(* Logix 5000 project; controller Project_Template vendor 1 type 14 code 106 rev 33.12; software revision 33.00 *)

TASK MainTask (continuous, watchdog 500 ms) : MainProgram

MODULES
   Local : vendor 1 type 14 code 106 (Compact 0, rev 33.12)
      Discrete_In_Slot_3 : 1769-IQ16 (Compact 3, rev 1.1, Input RPI 20 ms)
      Discrete_In_Slot_2 : 1769-IQ16 (Compact 2, rev 1.1, Input RPI 20 ms)
      Discrete_Out_Slot_4 : 1769-OW16 (Compact 4, rev 1.1, Output RPI 20 ms)
      ASCII_Slot_1 : vendor 1 type 109 code 66 (Compact 1, rev 2.1, Output RPI 100 ms)
      Discrete_Out_Slot_5 : 1769-OW16 (Compact 5, rev 1.1, Output RPI 20 ms)
END_MODULES

VAR_GLOBAL   (* controller tags *)
   AT_HOME : BOOL;
   AUTO : BOOL;
   end_start : BOOL;
   FLASH_FAST : BOOL := 1;
   Flash_Fast_Off : TIMER := (PRE := 250, ACC := 205, EN := 1, TT := 1);
   Flash_Fast_On : TIMER := (PRE := 250, ACC := 250, EN := 1, DN := 1);
   FLASH_MEDIUM : BOOL := 1;
   Flash_Medium_Off : TIMER := (PRE := 500, ACC := 467, EN := 1, TT := 1);
   Flash_Medium_On : TIMER := (PRE := 500, ACC := 500, EN := 1, DN := 1);
   FLASH_SLOW : BOOL;
   Flash_Slow_Off : TIMER := (PRE := 1000);
   Flash_Slow_On : TIMER := (PRE := 1000, ACC := 957, EN := 1, TT := 1);
   I_Auto_Mode_Selector : ALIAS FOR Local:2:I.Data.2;
   I_Barcode_Stop_Raised : ALIAS FOR Local:3:I.Data.1;
   I_Box_Ejector_Extended : ALIAS FOR Local:2:I.Data.4;
   I_Reject_Cyl_Lowered : ALIAS FOR Local:3:I.Data.2;
   I_Reset_PB : ALIAS FOR Local:2:I.Data.3;
   I_Start_PB : ALIAS FOR Local:2:I.Data.0;
   I_Stop_PB : ALIAS FOR Local:2:I.Data.1;
   I_Vacuum_Head_at_Conveyor : ALIAS FOR Local:3:I.Data.0;
   I_Vacuum_Head_at_Magazine : ALIAS FOR Local:2:I.Data.15;
   I_Vacuum_Head_Extended : ALIAS FOR Local:2:I.Data.14;
   I_Vacuum_Head_Lowered : ALIAS FOR Local:2:I.Data.10;
   I_Vacuum_Head_Raised : ALIAS FOR Local:2:I.Data.9;
   I_Vacuum_Head_Retracted : ALIAS FOR Local:2:I.Data.13;
   I_Vacuum_Head_Rotated_CCW : ALIAS FOR Local:2:I.Data.11;
   I_Vacuum_Head_Rotated_CW : ALIAS FOR Local:2:I.Data.12;
   I_Vacuum_Sensor_On : ALIAS FOR Local:3:I.Data.8;
   no_of_boxes : COUNTER := (PRE := 2);
   O_Amber_Tower_Ind : ALIAS FOR Local:5:O.Data.9;
   O_Barcode_Stop_Raise : ALIAS FOR Local:4:O.Data.14;
   O_Box_Eject : ALIAS FOR Local:4:O.Data.0;
   O_Conveyor_On : ALIAS FOR Local:5:O.Data.5;
   O_Green_Tower_Ind : ALIAS FOR Local:5:O.Data.8;
   O_Red_Tower_Ind : ALIAS FOR Local:5:O.Data.10;
   O_Reject_Cyl_Extend : ALIAS FOR Local:5:O.Data.0;
   O_Reject_Cyl_Lower : ALIAS FOR Local:4:O.Data.15;
   O_Vacuum_Head_Extend : ALIAS FOR Local:4:O.Data.8;
   O_Vacuum_Head_Lower : ALIAS FOR Local:4:O.Data.5;
   O_Vacuum_Head_Rotate_CCW : ALIAS FOR Local:4:O.Data.7;
   O_Vacuum_Head_Rotate_CW : ALIAS FOR Local:4:O.Data.6;
   O_Vacuum_Head_to_Conveyor : ALIAS FOR Local:4:O.Data.9;
   O_Vacuum_Head_to_Magazine : ALIAS FOR Local:4:O.Data.10;
   O_Vacuum_Off : ALIAS FOR Local:5:O.Data.2;
   O_Vacuum_On : ALIAS FOR Local:5:O.Data.1;
   Production_Step : DINT := 1792;
   proxy_stop : ALIAS FOR Local:3:I.Data.7;
   Raise_Vacuum : BOOL;
   Reset_Step : DINT;
   Retract_Box_Ejector : BOOL;
   Retract_Vacuum : BOOL;
   start_pb_count : COUNTER := (PRE := 1);
   Status_RESETTING : BOOL;
   Status_RUNNING : BOOL;
   Timer_Barcode_Delay : TIMER := (PRE := 1000, ACC := 1000, EN := 1, DN := 1);
   Timer_Conveyor_Delay : TIMER := (PRE := 3000, ACC := 492, EN := 1, TT := 1);
   Timer_Conveyor_Reset : TIMER := (PRE := 1000, ACC := 1000, EN := 1, DN := 1);
   timer_end_start : TIMER := (PRE := 1000);
   Timer_Extend_Delay : TIMER := (PRE := 1000);
   Timer_Production_Reset : TIMER := (PRE := 500);
   Timer_Reset : TIMER[7] := ([0].PRE := 250, [1].PRE := 250, [2].PRE := 250, [3].PRE := 250, [4].PRE := 250, [5].PRE := 250, [6].PRE := 250, [6].ACC := 250, [6].EN := 1, [6].DN := 1);
   Timer_Reset_Reset : TIMER := (PRE := 500);
   Timer_Vacuum : TIMER := (PRE := 250);
   Timer_Vacuum_Delay : TIMER := (PRE := 250);
END_VAR

PROGRAM MainProgram   (* main routine MainRoutine *)

ROUTINE a_Reset_Routine   (* ladder *)
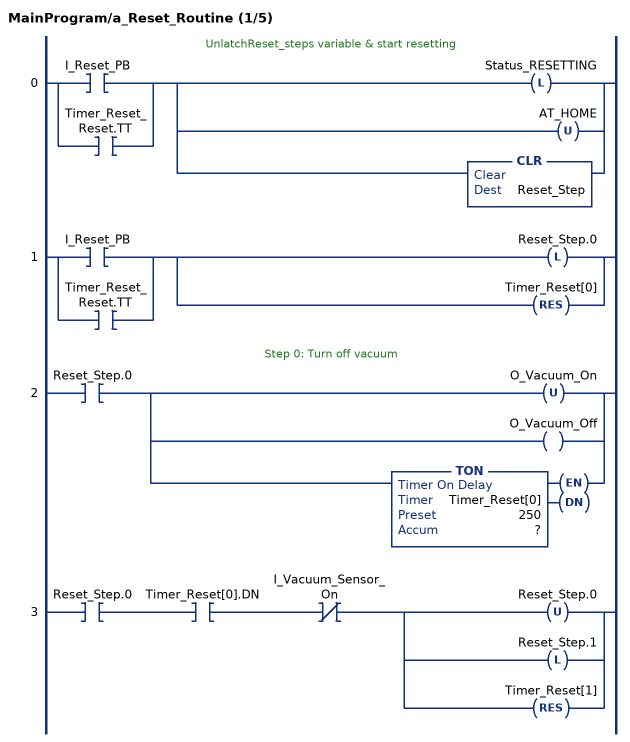
   // UnlatchReset_steps variable & start resetting
   0: [XIC(I_Reset_PB) ,XIC(Timer_Reset_Reset.TT) ][OTL(Status_RESETTING) ,OTU(AT_HOME) ,CLR(Reset_Step) ];
   1: [XIC(I_Reset_PB) ,XIC(Timer_Reset_Reset.TT) ][OTL(Reset_Step.0) ,RES(Timer_Reset[0]) ];
   // Step 0: Turn off vacuum
   2: XIC(Reset_Step.0)[OTU(O_Vacuum_On) ,OTE(O_Vacuum_Off) ,TON(Timer_Reset[0],?,?) ];
   3: XIC(Reset_Step.0)XIC(Timer_Reset[0].DN)XIO(I_Vacuum_Sensor_On)[OTU(Reset_Step.0) ,OTL(Reset_Step.1) ,RES(Timer_Reset[1]) ];
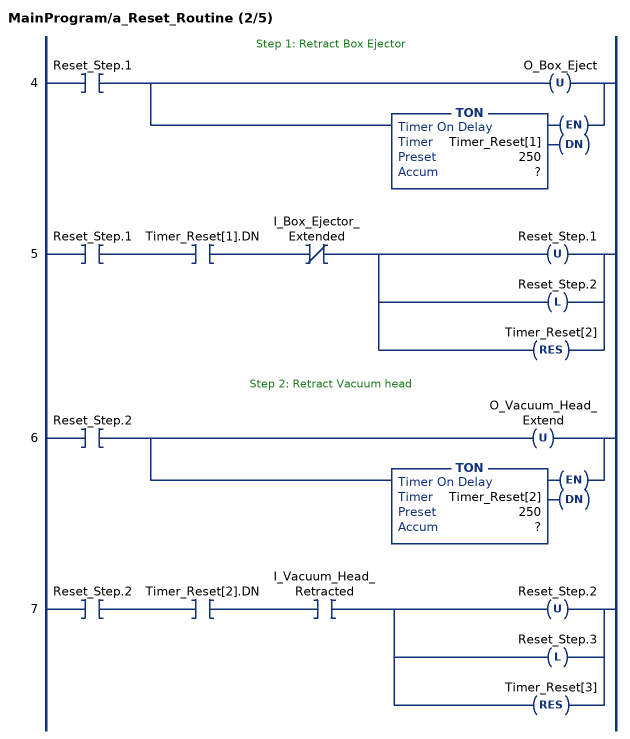
   // Step 1: Retract Box Ejector
   4: XIC(Reset_Step.1)[OTU(O_Box_Eject) ,TON(Timer_Reset[1],?,?) ];
   5: XIC(Reset_Step.1)XIC(Timer_Reset[1].DN)XIO(I_Box_Ejector_Extended)[OTU(Reset_Step.1) ,OTL(Reset_Step.2) ,RES(Timer_Reset[2]) ];
   // Step 2: Retract Vacuum head
   6: XIC(Reset_Step.2)[OTU(O_Vacuum_Head_Extend) ,TON(Timer_Reset[2],?,?) ];
   7: XIC(Reset_Step.2)XIC(Timer_Reset[2].DN)XIC(I_Vacuum_Head_Retracted)[OTU(Reset_Step.2) ,OTL(Reset_Step.3) ,RES(Timer_Reset[3]) ];
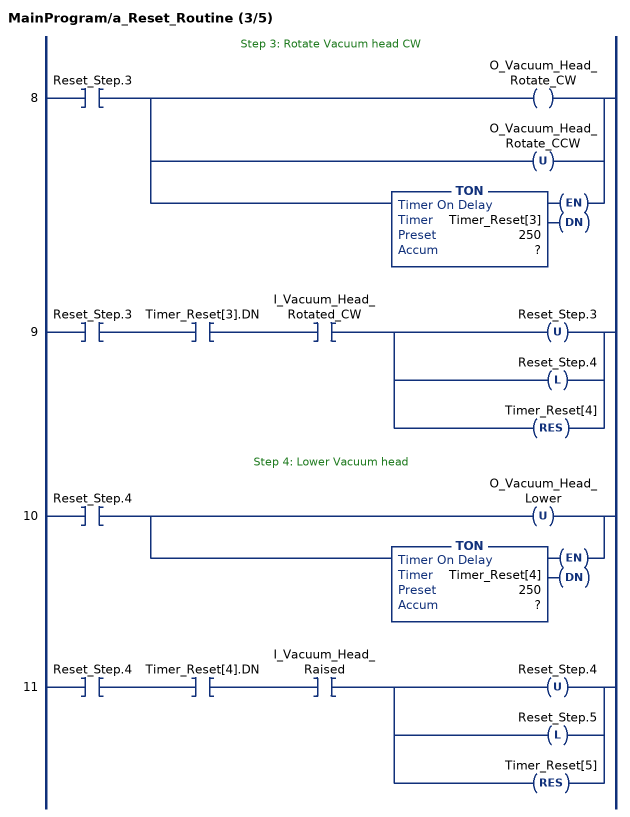
   // Step 3: Rotate Vacuum head CW
   8: XIC(Reset_Step.3)[OTE(O_Vacuum_Head_Rotate_CW) ,OTU(O_Vacuum_Head_Rotate_CCW) ,TON(Timer_Reset[3],?,?) ];
   9: XIC(Reset_Step.3)XIC(Timer_Reset[3].DN)XIC(I_Vacuum_Head_Rotated_CW)[OTU(Reset_Step.3) ,OTL(Reset_Step.4) ,RES(Timer_Reset[4]) ];
   // Step 4: Lower Vacuum head
   10: XIC(Reset_Step.4)[OTU(O_Vacuum_Head_Lower) ,TON(Timer_Reset[4],?,?) ];
   11: XIC(Reset_Step.4)XIC(Timer_Reset[4].DN)XIC(I_Vacuum_Head_Raised)[OTU(Reset_Step.4) ,OTL(Reset_Step.5) ,RES(Timer_Reset[5]) ];
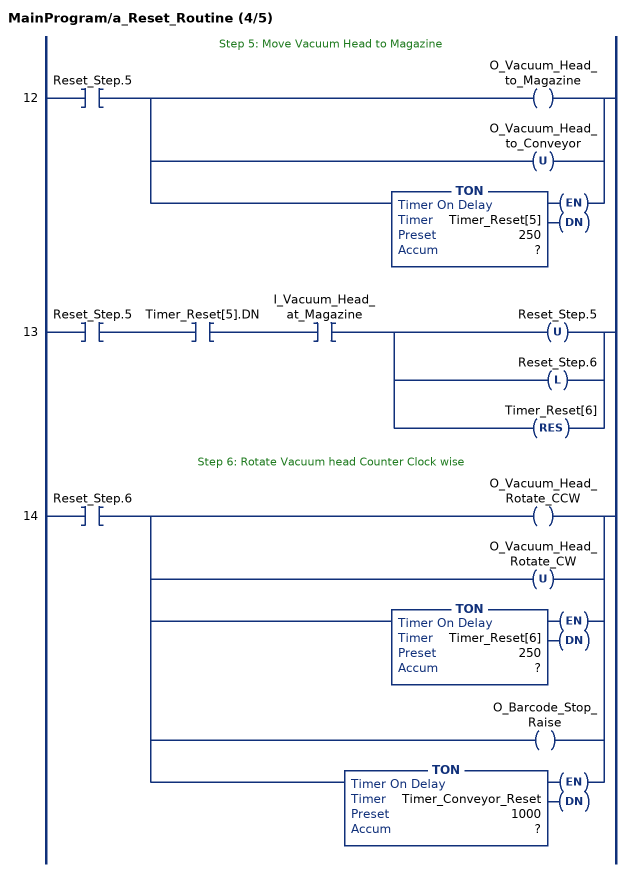
   // Step 5: Move Vacuum Head to Magazine
   12: XIC(Reset_Step.5)[OTE(O_Vacuum_Head_to_Magazine) ,OTU(O_Vacuum_Head_to_Conveyor) ,TON(Timer_Reset[5],?,?) ];
   13: XIC(Reset_Step.5)XIC(Timer_Reset[5].DN)XIC(I_Vacuum_Head_at_Magazine)[OTU(Reset_Step.5) ,OTL(Reset_Step.6) ,RES(Timer_Reset[6]) ];
   // Step 6: Rotate Vacuum head Counter Clock wise
   14: XIC(Reset_Step.6)[OTE(O_Vacuum_Head_Rotate_CCW) ,OTU(O_Vacuum_Head_Rotate_CW) ,TON(Timer_Reset[6],?,?) ,OTE(O_Barcode_Stop_Raise) ,TON(Timer_Conveyor_Reset,?,?) ];
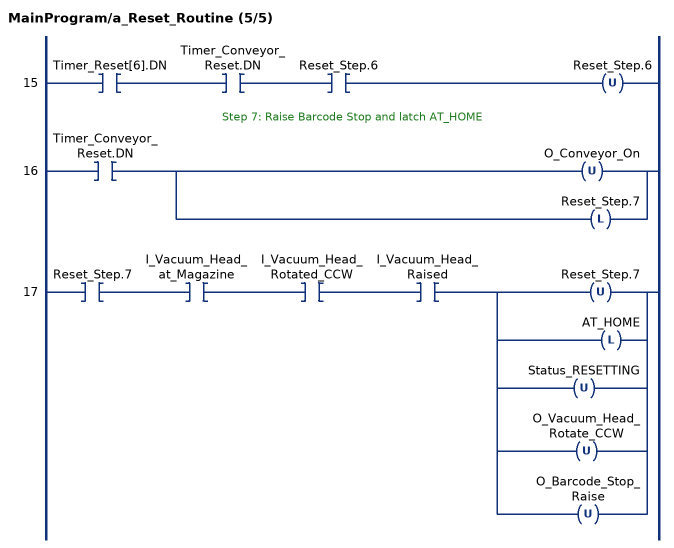
   15: XIC(Timer_Reset[6].DN)XIC(Timer_Conveyor_Reset.DN)XIC(Reset_Step.6)OTU(Reset_Step.6);
   // Step 7: Raise Barcode Stop and latch AT_HOME
   16: XIC(Timer_Conveyor_Reset.DN)[OTU(O_Conveyor_On) ,OTL(Reset_Step.7) ];
   17: XIC(Reset_Step.7)XIC(I_Vacuum_Head_at_Magazine)XIC(I_Vacuum_Head_Rotated_CCW)XIC(I_Vacuum_Head_Raised)[OTU(Reset_Step.7) ,OTL(AT_HOME) ,OTU(Status_RESETTING) ,OTU(O_Vacuum_Head_Rotate_CCW) ,OTU(O_Barcode_Stop_Raise) ];
END_ROUTINE

ROUTINE b_Production_Routine   (* ladder *)
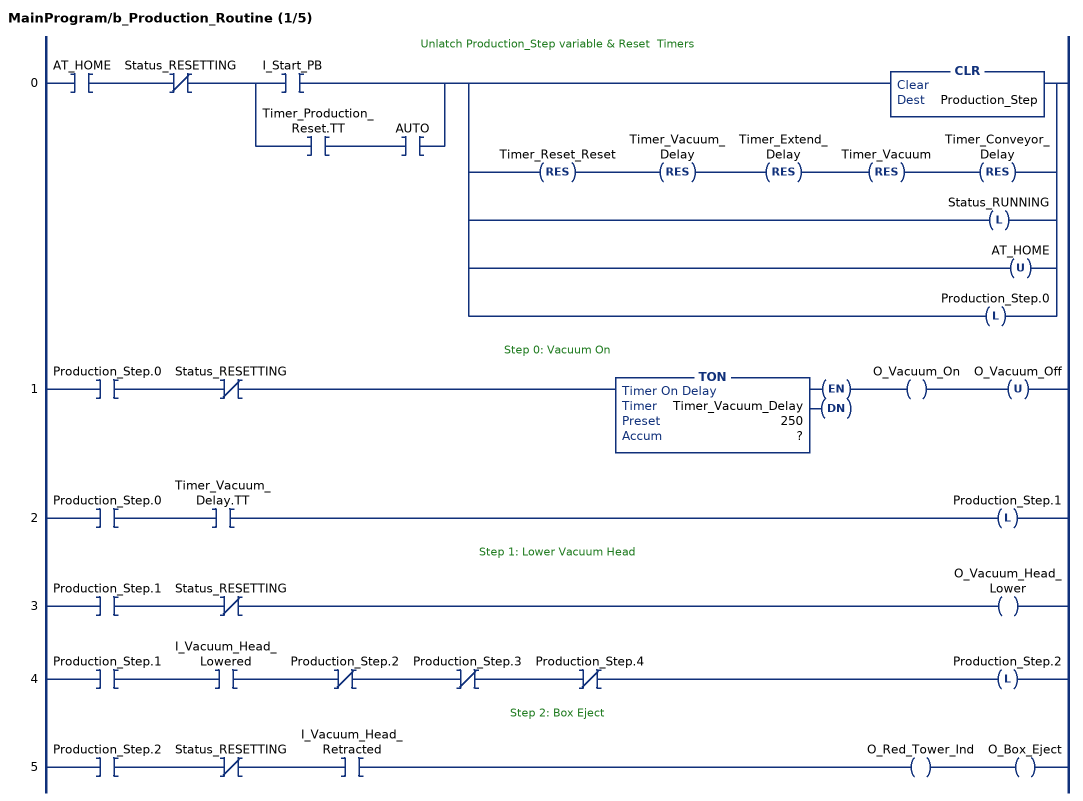
   // Unlatch Production_Step variable & Reset  Timers
   0: XIC(AT_HOME)XIO(Status_RESETTING)[XIC(I_Start_PB) ,XIC(Timer_Production_Reset.TT) XIC(AUTO) ][CLR(Production_Step) ,RES(Timer_Reset_Reset) RES(Timer_Vacuum_Delay) RES(Timer_Extend_Delay) RES(Timer_Vacuum) RES(Timer_Conveyor_Delay) ,OTL(Status_RUNNING) ,OTU(AT_HOME) ,OTL(Production_Step.0) ];
   // Step 0: Vacuum On
   1: XIC(Production_Step.0)XIO(Status_RESETTING)TON(Timer_Vacuum_Delay,?,?)OTE(O_Vacuum_On)OTU(O_Vacuum_Off);
   2: XIC(Production_Step.0)XIC(Timer_Vacuum_Delay.TT)OTL(Production_Step.1);
   // Step 1: Lower Vacuum Head
   3: XIC(Production_Step.1)XIO(Status_RESETTING)OTE(O_Vacuum_Head_Lower);
   4: XIC(Production_Step.1)XIC(I_Vacuum_Head_Lowered)XIO(Production_Step.2)XIO(Production_Step.3)XIO(Production_Step.4)OTL(Production_Step.2);
   // Step 2: Box Eject
   5: XIC(Production_Step.2)XIO(Status_RESETTING)XIC(I_Vacuum_Head_Retracted)OTE(O_Red_Tower_Ind)OTE(O_Box_Eject);
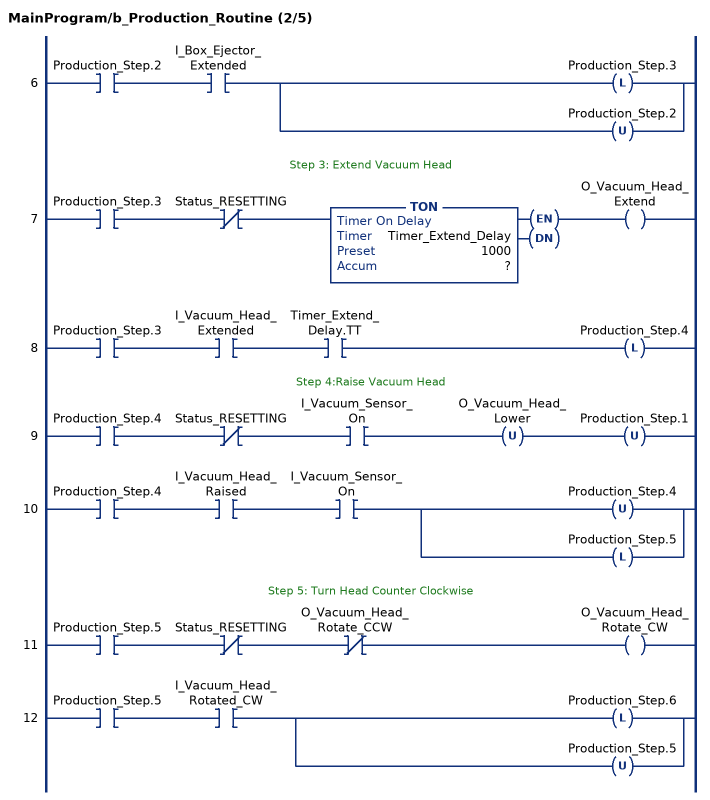
   6: XIC(Production_Step.2)XIC(I_Box_Ejector_Extended)[OTL(Production_Step.3) ,OTU(Production_Step.2) ];
   // Step 3: Extend Vacuum Head
   7: XIC(Production_Step.3)XIO(Status_RESETTING)TON(Timer_Extend_Delay,?,?)OTE(O_Vacuum_Head_Extend);
   8: XIC(Production_Step.3)XIC(I_Vacuum_Head_Extended)XIC(Timer_Extend_Delay.TT)OTL(Production_Step.4);
   // Step 4:Raise Vacuum Head
   9: XIC(Production_Step.4)XIO(Status_RESETTING)XIC(I_Vacuum_Sensor_On)OTU(O_Vacuum_Head_Lower)OTU(Production_Step.1);
   10: XIC(Production_Step.4)XIC(I_Vacuum_Head_Raised)XIC(I_Vacuum_Sensor_On)[OTU(Production_Step.4) ,OTL(Production_Step.5) ];
   // Step 5: Turn Head Counter Clockwise
   11: XIC(Production_Step.5)XIO(Status_RESETTING)XIO(O_Vacuum_Head_Rotate_CCW)OTE(O_Vacuum_Head_Rotate_CW);
   12: XIC(Production_Step.5)XIC(I_Vacuum_Head_Rotated_CW)[OTL(Production_Step.6) ,OTU(Production_Step.5) ];
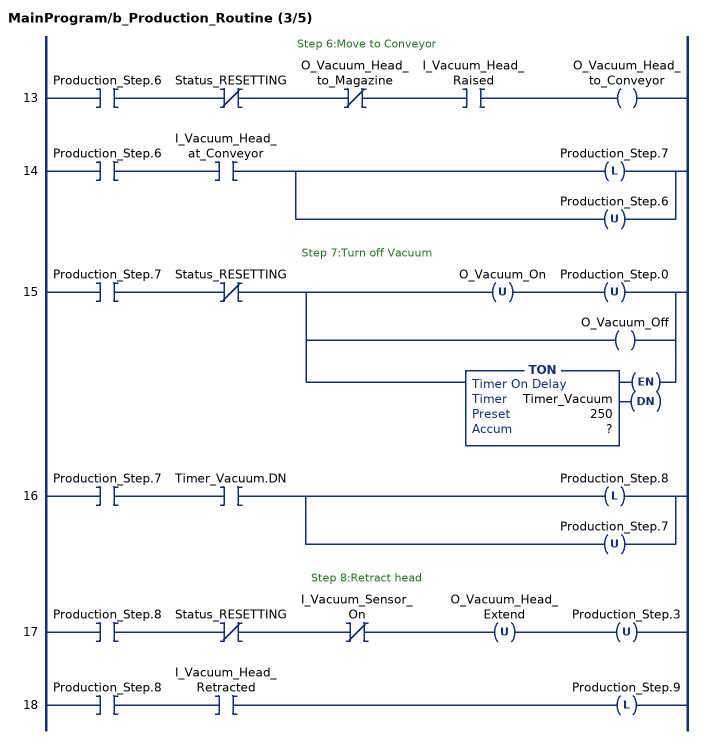
   // Step 6:Move to Conveyor
   13: XIC(Production_Step.6)XIO(Status_RESETTING)XIO(O_Vacuum_Head_to_Magazine)XIC(I_Vacuum_Head_Raised)OTE(O_Vacuum_Head_to_Conveyor);
   14: XIC(Production_Step.6)XIC(I_Vacuum_Head_at_Conveyor)[OTL(Production_Step.7) ,OTU(Production_Step.6) ];
   // Step 7:Turn off Vacuum
   15: XIC(Production_Step.7)XIO(Status_RESETTING)[OTU(O_Vacuum_On) OTU(Production_Step.0) ,OTE(O_Vacuum_Off) ,TON(Timer_Vacuum,?,?) ];
   16: XIC(Production_Step.7)XIC(Timer_Vacuum.DN)[OTL(Production_Step.8) ,OTU(Production_Step.7) ];
   // Step 8:Retract head
   17: XIC(Production_Step.8)XIO(Status_RESETTING)XIO(I_Vacuum_Sensor_On)OTU(O_Vacuum_Head_Extend)OTU(Production_Step.3);
   18: XIC(Production_Step.8)XIC(I_Vacuum_Head_Retracted)OTL(Production_Step.9);
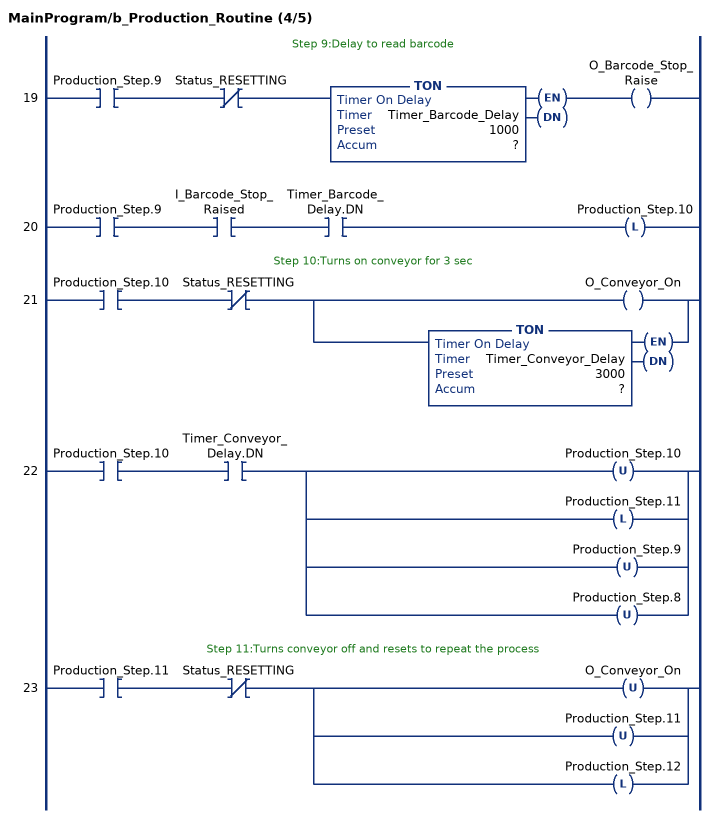
   // Step 9:Delay to read barcode
   19: XIC(Production_Step.9)XIO(Status_RESETTING)TON(Timer_Barcode_Delay,?,?)OTE(O_Barcode_Stop_Raise);
   20: XIC(Production_Step.9)XIC(I_Barcode_Stop_Raised)XIC(Timer_Barcode_Delay.DN)OTL(Production_Step.10);
   // Step 10:Turns on conveyor for 3 sec
   21: XIC(Production_Step.10)XIO(Status_RESETTING)[OTE(O_Conveyor_On) ,TON(Timer_Conveyor_Delay,?,?) ];
   22: XIC(Production_Step.10)XIC(Timer_Conveyor_Delay.DN)[OTU(Production_Step.10) ,OTL(Production_Step.11) ,OTU(Production_Step.9) ,OTU(Production_Step.8) ];
   // Step 11:Turns conveyor off and resets to repeat the process
   23: XIC(Production_Step.11)XIO(Status_RESETTING)[OTU(O_Conveyor_On) ,OTU(Production_Step.11) ,OTL(Production_Step.12) ];
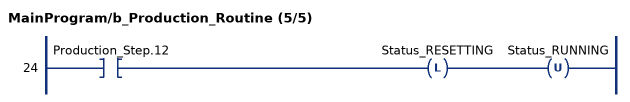
   24: XIC(Production_Step.12)OTL(Status_RESETTING)OTU(Status_RUNNING);
END_ROUTINE

ROUTINE MainRoutine   (* ladder *)
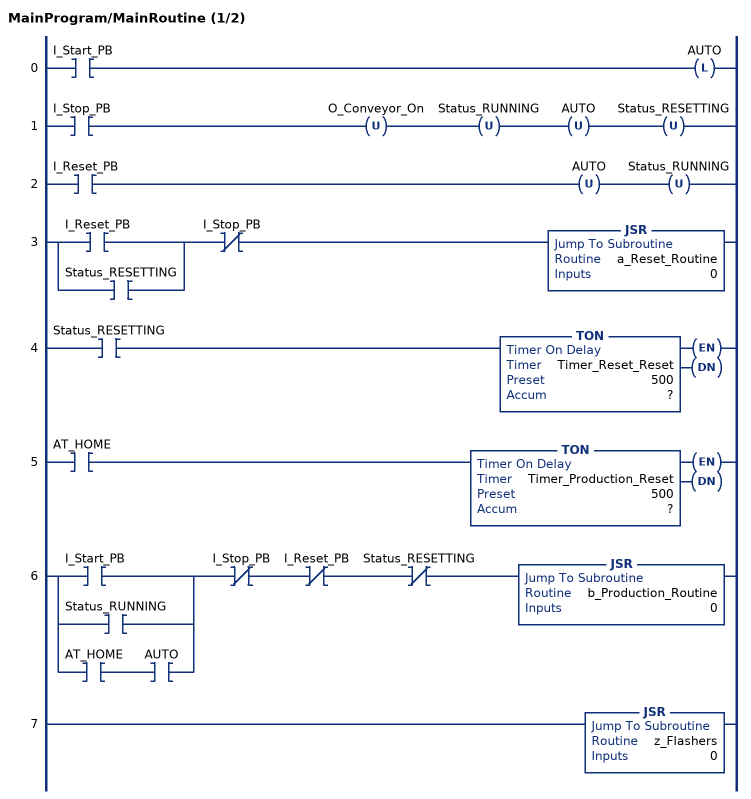
   0: XIC(I_Start_PB)OTL(AUTO);
   1: XIC(I_Stop_PB)OTU(O_Conveyor_On)OTU(Status_RUNNING)OTU(AUTO)OTU(Status_RESETTING);
   2: XIC(I_Reset_PB)OTU(AUTO)OTU(Status_RUNNING);
   3: [XIC(I_Reset_PB) ,XIC(Status_RESETTING) ]XIO(I_Stop_PB)JSR(a_Reset_Routine,0);
   4: XIC(Status_RESETTING)TON(Timer_Reset_Reset,?,?);
   5: XIC(AT_HOME)TON(Timer_Production_Reset,?,?);
   6: [XIC(I_Start_PB) ,XIC(Status_RUNNING) ,XIC(AT_HOME) XIC(AUTO) ]XIO(I_Stop_PB)XIO(I_Reset_PB)XIO(Status_RESETTING)JSR(b_Production_Routine,0);
   7: JSR(z_Flashers,0);
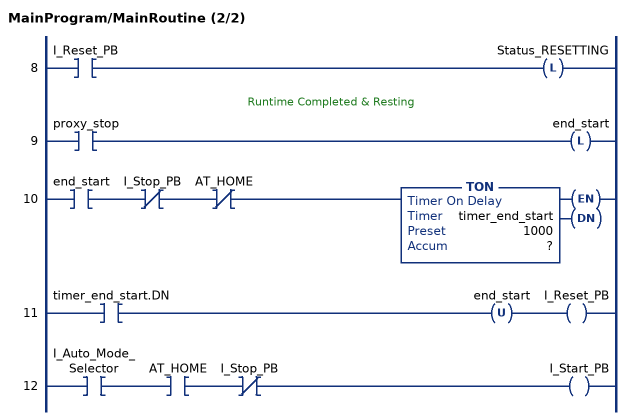
   8: XIC(I_Reset_PB)OTL(Status_RESETTING);
   // Runtime Completed & Resting
   9: XIC(proxy_stop)OTL(end_start);
   10: XIC(end_start)XIO(I_Stop_PB)XIO(AT_HOME)TON(timer_end_start,?,?);
   11 (stored rung type 1): XIC(timer_end_start.DN)OTU(end_start)OTE(I_Reset_PB);
   12: XIC(I_Auto_Mode_Selector)XIC(AT_HOME)XIO(I_Stop_PB)OTE(I_Start_PB);
END_ROUTINE

ROUTINE z_Flashers   (* ladder *)
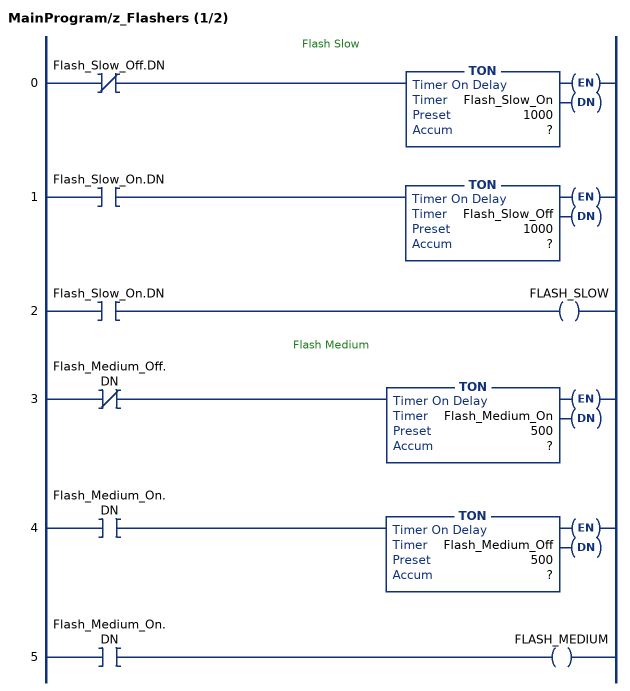
   // Flash Slow
   0: XIO(Flash_Slow_Off.DN)TON(Flash_Slow_On,?,?);
   1: XIC(Flash_Slow_On.DN)TON(Flash_Slow_Off,?,?);
   2: XIC(Flash_Slow_On.DN)OTE(FLASH_SLOW);
   // Flash Medium
   3: XIO(Flash_Medium_Off.DN)TON(Flash_Medium_On,?,?);
   4: XIC(Flash_Medium_On.DN)TON(Flash_Medium_Off,?,?);
   5: XIC(Flash_Medium_On.DN)OTE(FLASH_MEDIUM);
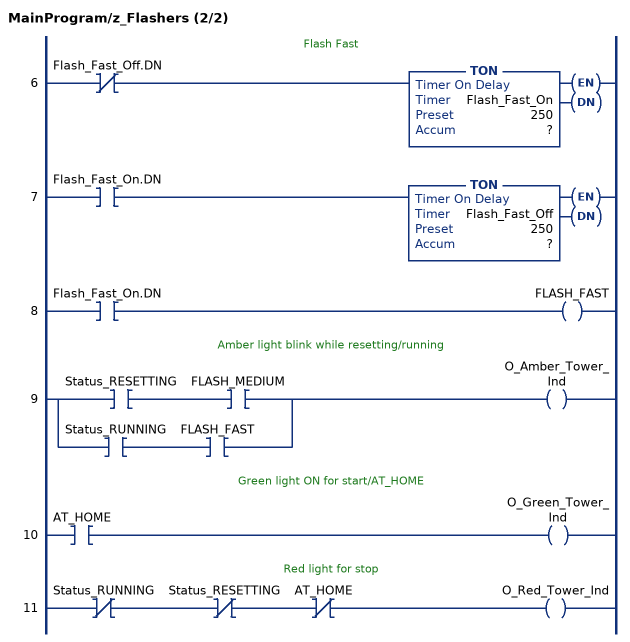
   // Flash Fast
   6: XIO(Flash_Fast_Off.DN)TON(Flash_Fast_On,?,?);
   7: XIC(Flash_Fast_On.DN)TON(Flash_Fast_Off,?,?);
   8: XIC(Flash_Fast_On.DN)OTE(FLASH_FAST);
   // Amber light blink while resetting/running
   9: [XIC(Status_RESETTING) XIC(FLASH_MEDIUM) ,XIC(Status_RUNNING) XIC(FLASH_FAST) ]OTE(O_Amber_Tower_Ind);
   // Green light ON for start/AT_HOME
   10: XIC(AT_HOME)OTE(O_Green_Tower_Ind);
   // Red light for stop
   11: XIO(Status_RUNNING)XIO(Status_RESETTING)XIO(AT_HOME)OTE(O_Red_Tower_Ind);
END_ROUTINE
END_PROGRAM
